// TwinCAT 3 PLC project testStepper
// ProgramVersion: 3.1.4023.0
// libraries:
//   Tc2_MC2, * (Beckhoff Automation GmbH)
//   Tc2_NC, * (Beckhoff Automation GmbH)
//   Tc2_Standard, * (Beckhoff Automation GmbH)
//   Tc2_System, * (Beckhoff Automation GmbH)
//   Tc3_Module, * (Beckhoff Automation GmbH)
//   VisuDialogs, * (System)
// project tree:
//   / GlobalTextList.TcGTLO (not stored), PlcTask.TcTTO (not stored), Visualization Manager.TcVMO (not stored)
//   GVLs/ GVL_AxisCtr.TcGVL (not stored), GVL_IO.TcGVL (not stored), GVL_NC.TcGVL
//   POUs/ DegreesToRelativeMovment.TcPOU (not stored), PositionToDegree.TcPOU (not stored), MAIN.TcPOU (not stored), POUNCPowerOn.TcPOU
//   VISUs/ testStepperVisu.TcVIS
// real-time tasks:
//   TASK PlcTask: cycle T#10ms, priority 20, ADS port 350
//   TASK PlcTask1: cycle T#10ms, priority 21, ADS port 351
// motion (NC):
//   TASK NC_test SAF: cycle T#2ms, priority 4, ADS port 501
//   TASK NC_test SVB: cycle T#10ms, priority 8, ADS port 511
//   AXIS Axis 1 (id 1)
//     OtherSettings: AllowMotionCmdToSlave=true
//     encoder EncType=1
//     drive DrvType=5
//       Analog: TorqueSetpointScale=10, ScaleFactorActTorque=0.1
//       TimeComp: TaskDelayCycles=1
//     controller CtrType=1
//       CtrPara: PriorControlFactor=1
//         Observer: BandWidth=20
// variable links:
//   testStepper/testStepper Instance <-> NC_test SAF/Axes/Axis 1
//     PlcTask Inputs/GVL_NC.stXAxis.NcToPlc <-> Outputs/ToPlc
//     PlcTask Outputs/GVL_NC.stXAxis.PlcToNc <-> Inputs/FromPlc

// ---- GVLs/GVL_NC.TcGVL
{attribute 'qualified_only'}
VAR_GLOBAL
	stXAxis :AXIS_REF;
	stXaxisStatus : ST_AxisStatus;
	
END_VAR

// ---- POUs/POUNCPowerOn.TcPOU
PROGRAM POUNCPowerOn
VAR
	fbXAxisPowerOn : MC_Power;
	fbXAxisDrive : MC_MoveRelative;
	DegreesToRelativeMovment_0: DegreesToRelativeMovment;
	movementBuffer : MC_BufferMode; 
	SetMaxRelativePoint : LREAL;
	SetMaxSteeringAngle : INT;
	inputAngle : INT;
	ExecuteMovement : BOOL;
	ExecuteMovement1 : BOOL;
	MC_MoveAbsolute_0: MC_MoveAbsolute;
	MC_Home_0: MC_Home;
	StartHoming: BOOL;
	endSW: BOOL;
	HomingActive: BOOL;
	MC_Reset_0: MC_Reset;
	reset: BOOL;
	PositionToDegree_0: PositionToDegree;
END_VAR

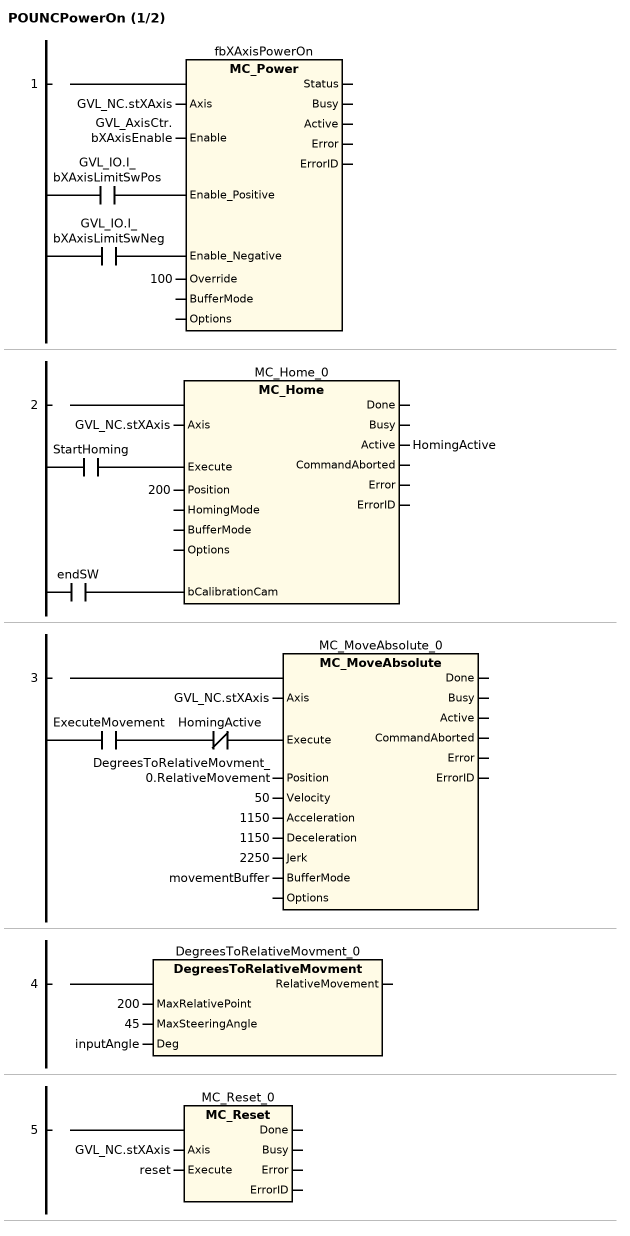
// NETWORK 1
fbXAxisPowerOn(
    Axis := GVL_NC.stXAxis,
    Enable := GVL_AxisCtr.bXAxisEnable,
    Enable_Positive := GVL_IO.I_bXAxisLimitSwPos,
    Enable_Negative := GVL_IO.I_bXAxisLimitSwNeg,
    Override := 100); // MC_Power

// NETWORK 2
MC_Home_0(
    Axis := GVL_NC.stXAxis,
    Execute := StartHoming,
    Position := 200,
    bCalibrationCam := endSW,
    Active => HomingActive); // MC_Home

// NETWORK 3
MC_MoveAbsolute_0(
    Axis := GVL_NC.stXAxis,
    Execute := ExecuteMovement AND NOT HomingActive,
    Position := DegreesToRelativeMovment_0.RelativeMovement,
    Velocity := 50,
    Acceleration := 1150,
    Deceleration := 1150,
    Jerk := 2250,
    BufferMode := movementBuffer); // MC_MoveAbsolute

// NETWORK 4
DegreesToRelativeMovment_0(MaxRelativePoint := 200, MaxSteeringAngle := 45, Deg := inputAngle); // DegreesToRelativeMovment

// NETWORK 5
MC_Reset_0(Axis := GVL_NC.stXAxis, Execute := reset); // MC_Reset

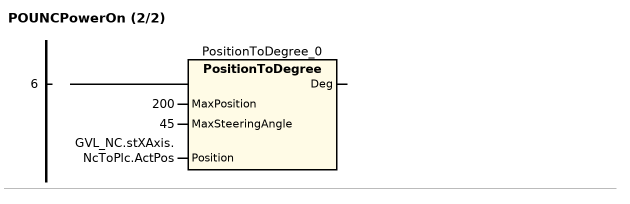
// NETWORK 6
PositionToDegree_0(MaxPosition := 200, MaxSteeringAngle := 45, Position := GVL_NC.stXAxis.NcToPlc.ActPos); // PositionToDegree

END_PROGRAM

// ---- VISUs/testStepperVisu.TcVIS
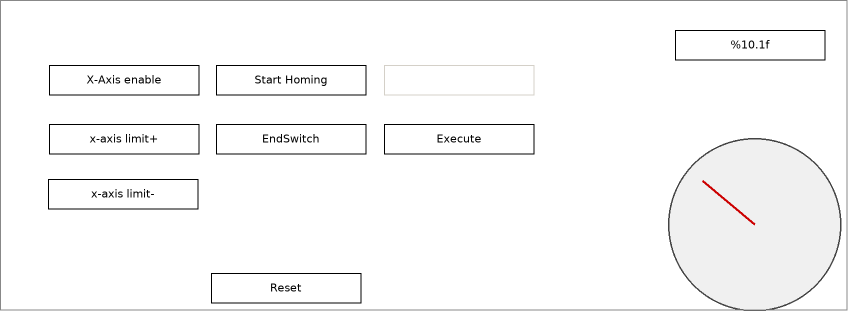
VISUALIZATION testStepperVisu  // 848x311
    Rectangle (49,65 150x30), "X-Axis enable"
        toggle GVL_AxisCtr.bXAxisEnable
    RoundedRectangle (49,124 150x30), "x-axis limit+", colour toggle: GVL_IO.I_bXAxisLimitSwPos
        toggle GVL_IO.I_bXAxisLimitSwPos
    RoundedRectangle (48,179 150x30), "x-axis limit-", colour toggle: GVL_IO.I_bXAxisLimitSwNeg
        toggle GVL_IO.I_bXAxisLimitSwNeg
    Rectangle (675,30 150x30), "%10.1f", text variable: GVL_NC.stXAxis.NcToPlc.ActPos
    Rectangle (384,124 150x30), "Execute"
        tap POUNCPowerOn.ExecuteMovement
    Rectangle (216,65 150x30), "Start Homing"
        tap POUNCPowerOn.StartHoming
    Rectangle (216,124 150x30), "EndSwitch"
        toggle POUNCPowerOn.endSW
    Rectangle (211,273 150x30), "Reset"
        tap POUNCPowerOn.reset
    Meter90 (661,138 187x173), value: POUNCPowerOn.PositionToDegree_0.Deg, style: Meter-Meter90-Gray, scale format: %.1f, scale -45..45
    Textfield (384,65 150x30)
        OnMouseDown: write POUNCPowerOn.inputAngle via InputWithLimits, min -45, max 45
END_VISUALIZATION
